// TIA Portal V20 export
// export: Created 2025-12-01T14:56:25.0333139Z, ExportSetting None, DisplayName Totally Integrated Automation Portal, DisplayVersion V20 Update 3, DisplayName TIA Portal Openness, DisplayVersion V20 Update 3, DisplayName TIA Portal Version Control Interface, DisplayVersion V20 Update 3, DisplayName STEP 7 Professional, DisplayVersion V20 Update 3, DisplayName STEP 7 Safety, DisplayVersion V20 Update 2, DisplayName WinCC Basic/Comfort/Advanced, DisplayVersion V20 Update 3, DisplayName WinCC Professional, DisplayVersion V20 Update 3, DisplayName WinCC Unified, DisplayVersion V20 Update 3
ORGANIZATION_BLOCK "OB1_Principal"   // OB1, LAD, ProgramCycle
TITLE = "Main Program Sweep (Cycle)"
{ S7_Optimized_Access := 'FALSE' }
AUTHOR : ESTANDAR
NAME : 20150525
VERSION : 3.1
// stored: AutoNumber false, SetENOAutomatically false
   VAR_TEMP
      OB1_EV_CLASS : Byte;   // Bits 0-3 = 1 (Coming event), Bits 4-7 = 1 (Event class 1)
      OB1_SCAN_1 : Byte;   // 1 (Cold restart scan 1 of OB 1), 3 (Scan 2-n of OB 1)
      OB1_PRIORITY : Byte;   // Priority of OB Execution
      OB1_OB_NUMBR : Byte;   // 1 (Organization block 1, OB1)
      OB1_RESERVED_1 : Byte;   // Reserved for system
      OB1_RESERVED_2 : Byte;   // Reserved for system
      OB1_PREV_CYCLE : Int;   // Cycle time of previous OB1 scan (milliseconds)
      OB1_MIN_CYCLE : Int;   // Minimum cycle time of OB1 (milliseconds)
      OB1_MAX_CYCLE : Int;   // Maximum cycle time of OB1 (milliseconds)
      OB1_DATE_TIME : Date_And_Time;   // Date and time OB1 started
      indice : UInt;
   END_VAR
   VAR_TEMP   // added for the SCL form of the ladder/FBD networks
      _w1 : Bool;
   END_VAR
BEGIN

REGION Network 1: Marcas Auxiliares CCPIF
   // *******************************************************************
   // * FUNCION: Generación marcas Auxiliares Generales del sistema     *
   // *******************************************************************
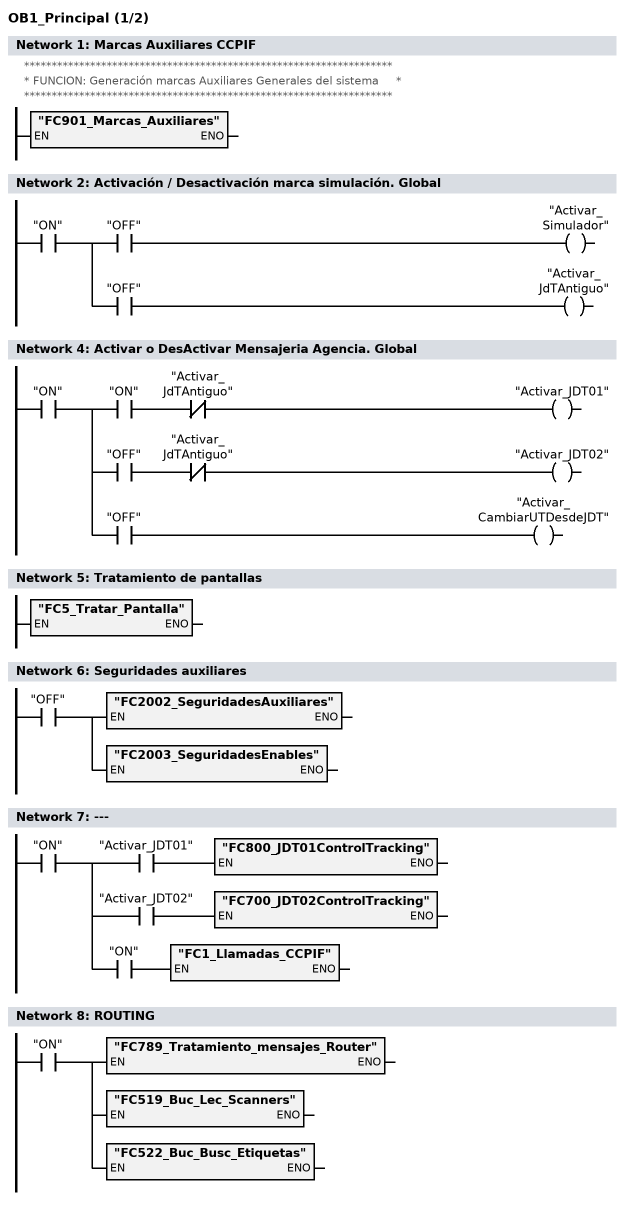
   RUNG wire#powerrail
      "FC901_Marcas_Auxiliares"()
   END_RUNG
   // the same network as SCL:
   "FC901_Marcas_Auxiliares"();
END_REGION

REGION Network 2: Activación / Desactivación marca simulación. Global
   RUNG wire#powerrail
      Contact( "ON" )
      wire#w1
      Contact( "OFF" )
      Coil( "Activar_Simulador" )
   END_RUNG
   RUNG wire#w1
      Contact( "OFF" )
      Coil( "Activar_JdTAntiguo" )
   END_RUNG
   // the same network as SCL:
   "Activar_Simulador" := "ON" AND "OFF";
   "Activar_JdTAntiguo" := "ON" AND "OFF";
END_REGION

NETWORK
TITLE = Cuando se desactive el JDT antiguo, tenemos que borrarnos todas las ordenes que se pudiesen quedar activas
// de lo contrario, habria problemas al realizar el cambio. Pablo
////////////////////////////////////////////////////////////////////////
////////////////////////////////////////////////////////////////////////
////////////////////////////////////////////////////////////////////////
/// --- Control de Cambio de Modo
      SET;
      A     "Activar_JdTAntiguo";
      FN    "Memo_JdTAntiguo_Desactivado";
      JC    BorradoDatos_CambioModo;

      SET;
      A     "Activar_JdTAntiguo";
      FP    "Memo_JdTAntiguo_Activado";
      JC    BorradoDatos_CambioModo;

      JU    Fin_CambioModo;

////////////////////////////////////////////////////////////////////////
////////////////////////////////////////////////////////////////////////
////////////////////////////////////////////////////////////////////////
/// --- Borrado de Datos
BorradoDatos_CambioModo:NOP   0;
      SET;
      S     "DB801_JDT01StatusCOM".ResetBD;
      S     "DB701_JDT02StatusCOM".ResetBD;


////////////////////////////////////////////////////////////////////////
////////////////////////////////////////////////////////////////////////
////////////////////////////////////////////////////////////////////////
/// --- Final de Cambio de Modo
Fin_CambioModo:NOP   0;



REGION Network 4: Activar o DesActivar Mensajeria Agencia. Global
   RUNG wire#powerrail
      Contact( "ON" )
      wire#w1
      Contact( "ON" )
      I_Contact( "Activar_JdTAntiguo" )
      Coil( "Activar_JDT01" )
   END_RUNG
   RUNG wire#w1
      Contact( "OFF" )
      I_Contact( "Activar_JdTAntiguo" )
      Coil( "Activar_JDT02" )
   END_RUNG
   RUNG wire#w1
      Contact( "OFF" )
      Coil( "Activar_CambiarUTDesdeJDT" )
   END_RUNG
   // the same network as SCL:
   "Activar_JDT01" := "ON" AND "ON" AND NOT "Activar_JdTAntiguo";
   "Activar_JDT02" := "ON" AND "OFF" AND NOT "Activar_JdTAntiguo";
   "Activar_CambiarUTDesdeJDT" := "ON" AND "OFF";
END_REGION

REGION Network 5: Tratamiento de pantallas
   RUNG wire#powerrail
      "FC5_Tratar_Pantalla"()
   END_RUNG
   // the same network as SCL:
   "FC5_Tratar_Pantalla"();
END_REGION

REGION Network 6: Seguridades auxiliares
   RUNG wire#powerrail
      Contact( "OFF" )
      wire#w1
      "FC2002_SeguridadesAuxiliares"()
   END_RUNG
   RUNG wire#w1
      "FC2003_SeguridadesEnables"()
   END_RUNG
   // the same network as SCL:
   #_w1 := "OFF";
   IF #_w1 THEN
       "FC2002_SeguridadesAuxiliares"();
       "FC2003_SeguridadesEnables"();
   END_IF;
END_REGION

REGION Network 7: ---
   RUNG wire#powerrail
      Contact( "ON" )
      wire#w1
      Contact( "Activar_JDT01" )
      "FC800_JDT01ControlTracking"()
   END_RUNG
   RUNG wire#w1
      Contact( "Activar_JDT02" )
      "FC700_JDT02ControlTracking"()
   END_RUNG
   RUNG wire#w1
      Contact( "ON" )
      "FC1_Llamadas_CCPIF"()
   END_RUNG
   // the same network as SCL:
   #_w1 := "ON";
   IF "ON" AND "Activar_JDT01" THEN "FC800_JDT01ControlTracking"(); END_IF;
   IF #_w1 AND "Activar_JDT02" THEN "FC700_JDT02ControlTracking"(); END_IF;
   IF #_w1 AND "ON" THEN "FC1_Llamadas_CCPIF"(); END_IF;
END_REGION

REGION Network 8: ROUTING
   RUNG wire#powerrail
      Contact( "ON" )
      wire#w1
      "FC789_Tratamiento_mensajes_Router"()
   END_RUNG
   RUNG wire#w1
      "FC519_Buc_Lec_Scanners"()
   END_RUNG
   RUNG wire#w1
      "FC522_Buc_Busc_Etiquetas"()
   END_RUNG
   // the same network as SCL:
   #_w1 := "ON";
   IF #_w1 THEN
       "FC789_Tratamiento_mensajes_Router"();
       "FC519_Buc_Lec_Scanners"();
       "FC522_Buc_Busc_Etiquetas"();
   END_IF;
END_REGION

REGION Network 9: Llamadas CBOXES
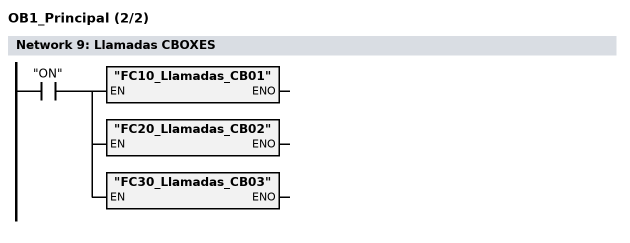
   RUNG wire#powerrail
      Contact( "ON" )
      wire#w1
      "FC10_Llamadas_CB01"()
   END_RUNG
   RUNG wire#w1
      "FC20_Llamadas_CB02"()
   END_RUNG
   RUNG wire#w1
      "FC30_Llamadas_CB03"()
   END_RUNG
   // the same network as SCL:
   #_w1 := "ON";
   IF #_w1 THEN
       "FC10_Llamadas_CB01"();
       "FC20_Llamadas_CB02"();
       "FC30_Llamadas_CB03"();
   END_IF;
END_REGION

NETWORK
TITLE = Configuracion de Mesas >> Activar JDT Antiguo
///////////////////////////////////////////////////////////////////////////
///////////////////////////////////////////////////////////////////////////
///////////////////////////////////////////////////////////////////////////
/// Configuracion de Mesas >> Activar JDT Antiguo
      SET;
      AN    "Activar_JdTAntiguo";
      JC    FinalConfigMesas;


///////////////////////////////////////////////////////////////////////////
/// DeActivar Error De Datos
      L     1;
      T     #indice;

InicioBucle_ConfigMesas:NOP   0;
      SET;
      =     "DB850_DefinicionMesas".Mesa[#indice].ConfigMesa.SinErrorDeDatosCargada;
      =     "DB850_DefinicionMesas".Mesa[#indice].ConfigMesa.SinErrorDeDatosVacia;

      L     #indice;
      L     1;
      +I;
      T     #indice;

      L     #indice;
      L     "CTE_MaxMesas";
      >I;
      JC    FinalConfigMesas;
      JU    InicioBucle_ConfigMesas;


///////////////////////////////////////////////////////////////////////////
///////////////////////////////////////////////////////////////////////////
///////////////////////////////////////////////////////////////////////////
/// Final de Configuracion de Mesas >> Activar JDT Antiguo
FinalConfigMesas:NOP   0;


END_ORGANIZATION_BLOCK
